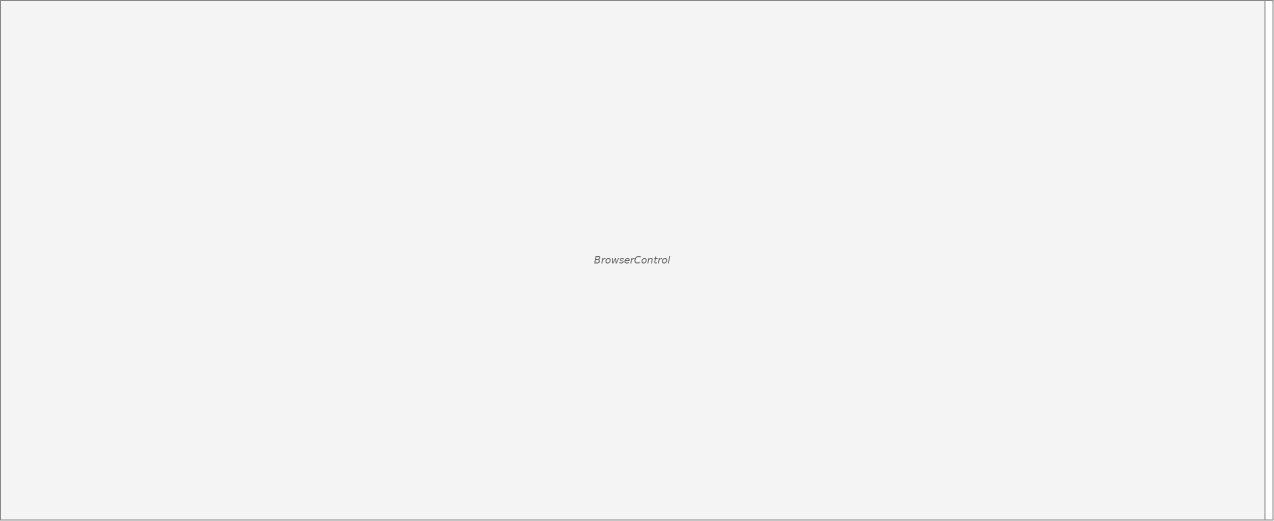
VISUALIZATION GraphScreen  // 1274x521
    BrowserControl (0,0 1265x520)
        p3734058945: GVL.graphURL
END_VISUALIZATION

(* stored: Version 1.1.0.1, ProductVersion 3.1.4022.18
   Visu GraphScreen: Id {c82a5f96-6d6e-4979-a04e-fa6429e6ff8c} *)
